// TIA Portal V17 export
// export: Created 2022-07-20T06:59:48.9463135Z, ExportSetting WithDefaults, DisplayName Totally Integrated Automation Portal, DisplayVersion V17, DisplayName TIA Portal Openness, DisplayVersion V17, DisplayName TIA Portal Version Control Interface, DisplayVersion V17, DisplayName SINAMICS Startdrive Advanced, DisplayVersion V17, DisplayName SINAMICS Startdrive G130, G150, S120, S150, SINAMICS MV, S210, DisplayVersion V17, DisplayName SINAMICS Startdrive G110M, G120, G120C, G120D, G120P, G115D, DisplayVersion V17, DisplayName STEP 7 Professional, DisplayVersion V17, DisplayName STEP 7 Safety, DisplayVersion V17, DisplayName WinCC Advanced, DisplayVersion V17
FUNCTION_BLOCK "FB10223_CoveredDistanceCounter"   // FB10223, LAD
{ S7_Optimized_Access := 'TRUE' }
VERSION : 0.1
// stored: AutoNumber false, IsIECCheckEnabled false, IsRetainMemResEnabled false, MemoryReserve 100, SetENOAutomatically false, UDAEnableTagReadback false
   VAR_INPUT
      ActualPosition : LReal;
   END_VAR
   VAR_IN_OUT
      ResetCounter : Bool;
      CoveredDistance : LReal;
   END_VAR
   VAR
      R_TRIG_PositionChanged : R_TRIG;
   END_VAR
   VAR RETAIN
      PreviousPosition : LReal;
   END_VAR
BEGIN

REGION Network 1 (SCL): Edge Signals & Timers Manegement
   REGION EDGE SIGNALS
       #R_TRIG_PositionChanged(CLK := ABS(#ActualPosition - #PreviousPosition) > 1.0);
   END_REGION
END_REGION

REGION Network 2 (SCL): Counter Management
   IF #R_TRIG_PositionChanged.Q THEN
       #CoveredDistance += ABS(#ActualPosition - #PreviousPosition);
       #PreviousPosition := #ActualPosition;
   ELSIF #ResetCounter THEN
       #CoveredDistance := 0.0;
       IF #CoveredDistance = 0.0 THEN
           #ResetCounter := FALSE;
       END_IF;
   END_IF;
END_REGION
END_FUNCTION_BLOCK
